Staubli VAL3: AfterWorkPlace.pgx

public program AfterWorkPlace(num x_nWorkplaceIn)
begin
  //参数：x_nWorkplaceIn 工位参数，传入的参数是 DataBase:nWorkPlaceIndex
  //引用位置:Teach:Prodcut.pgx
  //功能：工位完成后，机器人已经回到零位。一般可以输出IO
  //备注：


  //  if bDebug
  //    popUpMsg("AfterWorkPlace")
  //    logMsg("AfterWorkPlace")
  //
  //
  //  endIf



end
